Staubli VAL3: sendToNextRobot.pgx

public program sendToNextRobot(sio x_sSocketClient (dimensions=1), num x_nTimeOut (dimensions=1), num x_nID (dimensions=1), trsf x_trObjectPos (dimensions=1), num x_nLatchedValue (dimensions=1), num& x_nError (dimensions=1))
  local num l_i
  local num l_nAsciiCode
  local num l_nClock
  local num l_nNumCharRead
  local num l_nNumCharWrite
  local string l_sCharRead
  local string l_sString
begin
  // This program sends a telegram via a socket client.
  // The telegram contains all the information of a detected object,
  //  this information is meant to be used by a detection library of
  //  another robot. The detection library "Socket" uses this information.
  // The format of the telegram is:
  //  {ID=i,X=x.xxx,Y=y.yyy,RZ=r.rrr,L=l.llllll}, where "{" is the initial
  //  character, "i" is the ID of the detected object, "x.xxx" is the
  //  value on X, "y.yyy" is the value on Y, "r.rrr" is the value on
  //  RZ, "l.llllll" is the latched encoder value, "," is the separator
  //  character and "}" is the end character. At the end, it waits for the
  //  character "$" as confirmation of good reception.
  //
  // Input Param
  //  x_sSocketClient : Socket client used to send the message.
  //  x_nTimeOut      : Timeout for the socket client to read/write one
  //                     character.
  //  x_nID           : ID of the detected object.
  //  x_trObjectPos   : Transformation of the detected object.
  //  x_nEncLatchVal  : Latched encoder value of the detected object.
  //
  // Output Param
  //  x_nError        :
  //                0 = No error, message sent.
  //                1 = The socket sent as a parameter is not working.
  //                     Bad link or device in error.
  //                2 = Message not sent. Timeout expired. The other robot
  //                     is not present on the network.
  //                3 = Timeout expired. The other robot is not working
  //                     with the detection library "Socket".
  //                4 = Message sent but the server from the other robot
  //                     didn't acknowledge reception before expiration
  //                     of timeout.
  //
  //----------------------------------------------------------------
  //
  x_nError=0
  //
  // Check if the socket "sent as a parameter is working.
  if ioStatus(x_sSocketClient)<0
    x_nError=1
    popUpMsg(lang:sListOfMessage[63])
    if bAnd(cfg:nLog,cfg:nLOGMISC)==cfg:nLOGMISC
      ? "MOT(sendToNextRobot)>> "+lang:sListOfMessage[63]
    endIf
    return
  endIf
  //
  // Defines the timeout on the socket.
  sioCtrl(x_sSocketClient,"timeout",x_nTimeOut)
  // Test if the other robot is connected to the network and if the
  //  application is running with the detection library "Socket".
  l_nNumCharWrite=sioSet(x_sSocketClient,13)
  if l_nNumCharWrite==-1
    // Timeout expired. The other robot is not present on the network.
    x_nError=2
    popUpMsg(lang:sListOfMessage[64])
    if bAnd(cfg:nLog,cfg:nLOGMISC)==cfg:nLOGMISC
      ? "MOT(sendToNextRobot)>> "+lang:sListOfMessage[64]
    endIf
    return
  elseIf l_nNumCharWrite==0
    // Timeout expired. The other robot is not working with the detection
    //  library "Socket".
    x_nError=3
    popUpMsg(lang:sListOfMessage[65])
    if bAnd(cfg:nLog,cfg:nLOGMISC)==cfg:nLOGMISC
      ? "MOT(sendToNextRobot)>> "+lang:sListOfMessage[65]
    endIf
    clearBuffer(x_sSocketClient)
    return
  endIf
  // After re-launching the application on the other robot, a few extra
  //  character are needed to establish a good connection.
  for l_i=1 to 5
    l_nNumCharWrite=sioSet(x_sSocketClient,13)
  endFor
  //
  // Builds up telegram.
  l_sString="{ID="
  l_sString=l_sString+toString("",x_nID)
  l_sString=l_sString+",X="
  l_sString=l_sString+toString(".3",x_trObjectPos.x)
  l_sString=l_sString+",Y="
  l_sString=l_sString+toString(".3",x_trObjectPos.y)
  l_sString=l_sString+",RZ="
  l_sString=l_sString+toString(".3",x_trObjectPos.rz)
  l_sString=l_sString+",L="
  l_sString=l_sString+toString(".6",x_nLatchedValue)
  l_sString=l_sString+"}"
  //
  // Sends telegram character by character.
  for l_i=0 to len(l_sString)-1
    l_nNumCharWrite=sioSet(x_sSocketClient,asc(l_sString,l_i))
    if l_nNumCharWrite==-1
      // Timeout expired. The other robot is not present on the network.
      x_nError=2
      popUpMsg(lang:sListOfMessage[64])
      if bAnd(cfg:nLog,cfg:nLOGMISC)==cfg:nLOGMISC
        ? "MOT(sendToNextRobot)>> "+lang:sListOfMessage[64]
      endIf
      return
    elseIf l_nNumCharWrite==0
      // Timeout expired. The other robot is not working with the detection
      //  library "Socket".
      x_nError=3
      popUpMsg(lang:sListOfMessage[65])
      if bAnd(cfg:nLog,cfg:nLOGMISC)==cfg:nLOGMISC
        ? "MOT(sendToNextRobot)>> "+lang:sListOfMessage[65]
      endIf
      clearBuffer(x_sSocketClient)
      return
    endIf
  endFor
  //
  // Waits for character "confirmation of good reception".
  l_sCharRead=""
  do
    // Reads one character from socket
    l_nNumCharRead=sioGet(x_sSocketClient,l_nAsciiCode)
    // If one character read
    if l_nNumCharRead==1
      l_sCharRead=chr(l_nAsciiCode)
    else
      // The server from the other robot didn't acknowledge reception
      //  before expiration of timeout.
      x_nError=4
      popUpMsg(lang:sListOfMessage[66])
      if bAnd(cfg:nLog,cfg:nLOGMISC)==cfg:nLOGMISC
        ? "MOT(sendToNextRobot)>> "+lang:sListOfMessage[66]
      endIf
      return
    endIf
  until l_sCharRead=="$"
  //
  if bAnd(cfg:nLog,cfg:nLOGMISC)==cfg:nLOGMISC
    ? "MOT(sendToNextRobot)>> Message sent: "
    ? l_sString
  endIf
  //
end
